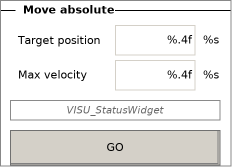
VISUALIZATION VISU_BaseAxis_MoveAbsolute  // 232x167
VAR_IN_OUT
	axis : BaseAxis;
    axisWidget : BaseAxisWidget;
    positionSymbol : STRING;
    velocitySymbol : STRING;
END_VAR
    Label (15,26 100x29), "Target position"
    Button (10,130 210x35), "GO", input disabled if: axis.processes.moveAbsolute.statuses.enabledStatus.disabled
        OnMouseClick: execute { axis.processes.moveAbsolute.do_request := TRUE; }
    Textfield (115,60 80x30), "%.4f", text variable: axis.processes.moveAbsolute.set.maxVelocity, input disabled if: axis.processes.moveAbsolute.statuses.enabledStatus.disabled
        OnMouseClick: write the text variable via VisuDialogs.Numpad
    Label (15,60 100x30), "Max velocity"
    Line (0,10) (15,10)
    Label (20,0 150x20), "Move absolute"
    Line (115,10) (230,10)
    Textfield (115,25 80x30), "%.4f", text variable: axis.processes.moveAbsolute.set.position, input disabled if: axis.processes.moveAbsolute.statuses.enabledStatus.disabled
        OnMouseClick: write the text variable via VisuDialogs.Numpad
    Frame (10,100 210x20)
        shows VISU_StatusWidget(widget := axisWidget.moveAbsoluteProcess.actualStatus)
    Rectangle (200,25 30x30), "%s", text variable: positionSymbol
    Rectangle (200,60 30x30), "%s", text variable: velocitySymbol
END_VISUALIZATION

(* stored: Version 1.1.0.1, ProductVersion 3.1.4019.2
   Visu VISU_BaseAxis_MoveAbsolute: Id {f2e1597b-ef2f-490c-a34b-3a4646c47e9c} *)
